// TwinCAT 3 PLC project PLC
// ProgramVersion: 3.1.4024.0
// libraries:
//   SPT Base Types, * (Beckhoff Automation LLC)
//   SPT Motion Control, * (Beckhoff Automation LLC)
//   Tc2_MC2, * (Beckhoff Automation GmbH)
//   Tc2_MC2_Drive, * (Beckhoff Automation GmbH)
//   Tc2_Standard, * (Beckhoff Automation GmbH)
//   Tc2_System, * (Beckhoff Automation GmbH)
//   Tc3_Module, * (Beckhoff Automation GmbH)
// project tree:
//   DUTs/ MoveState_t.TcDUT
//   GVLs/ IO.TcGVL (not stored), SafetyGlobalVariableList.TcGVL (not stored)
//   / PlcTask.TcTTO, SafetyTask.TcTTO
//   POUs/ MAIN.TcPOU (not stored), TestAxis1.TcPOU, SAFETY.TcPOU (not stored), TestAxis2.TcPOU
// real-time tasks:
//   TASK PlcTask: cycle T#10ms, priority 20, ADS port 350
//   TASK SafetyTask: cycle T#10ms, priority 21, ADS port 351
// motion (NC):
//   TASK NC-Task SAF: cycle T#2ms, priority 4, ADS port 501
//   TASK NC-Task SVB: cycle T#10ms, priority 8, ADS port 511
//   AXIS Axis 1 (id 1)
//     Dynamic: Acceleration=3272.24, Deceleration=3272.24, Jerk=9816.73
//     Velo: RefSearch=21.81495, RefSync=21.81495, SlowManual=109.07475, FastManual=654.4485, Fast=2181.495, Maximum=2181.49
//     PositionAreaControl: Enable=false, Range=1000
//     TargetPosControl: Enable=false, Range=1000
//     OtherSettings: AllowMotionCmdToSlave=true
//     encoder EncType=8
//       EncPara: ScaleFactorNumerator=60, ScaleFactorDenominator=1048576, MaxCount=#xffffffff
//     drive DrvType=9
//       DrvPara: MaxCount=#xffffffff, DriveControlDWord=#x00030100
//         Analog: VeloReferenz=2399.6445, VeloScale=1.02400649589962, TorqueSetpointScale=10, ScaleFactorActTorque=0.1
//         TimeComp: TaskDelayCycles=1
//     controller CtrType=1
//       CtrPara: PriorControlFactor=1
//         PosDiffControl: Enable=false, Range=15
//         Observer: BandWidth=20
//   AXIS Axis 2 (id 2)
//     Dynamic: Acceleration=3272.24, Deceleration=3272.24, Jerk=9816.73
//     Velo: RefSearch=21.81495, RefSync=21.81495, SlowManual=109.07475, FastManual=654.4485, Fast=2181.495, Maximum=2181.49
//     PositionAreaControl: Enable=false, Range=1000
//     TargetPosControl: Enable=false, Range=1000
//     OtherSettings: AllowMotionCmdToSlave=true
//     encoder EncType=8
//       EncPara: ScaleFactorNumerator=60, ScaleFactorDenominator=1048576, MaxCount=#xffffffff
//     drive DrvType=9
//       DrvPara: MaxCount=#xffffffff, DriveControlDWord=#x00030100
//         Analog: VeloReferenz=2399.6445, VeloScale=1.02400649589962, TorqueSetpointScale=10, ScaleFactorActTorque=0.1
//         TimeComp: TaskDelayCycles=1
//     controller CtrType=1
//       CtrPara: PriorControlFactor=1
//         PosDiffControl: Enable=false, Range=15
//         Observer: BandWidth=20
// I/O:
//   DEVICE CP6700-0001-0050, AmsNetId 5.81.155.22.4.1
//     Term 1 (EK1100) [EK1100 EtherCAT Coupler (2A E-Bus)]
//       Term 2 (EL1008) [EL1008 8Ch. Dig. Input 24V, 3ms]
//       Term 3 (EL1008) [EL1008 8Ch. Dig. Input 24V, 3ms]
//       Term 4 (EL2008) [EL2008 8Ch. Dig. Output 24V, 0.5A]
//       Term 5 (EL6910) [EL6910, TwinSAFE PLC]
//       Term 6 (EL1918) [EL1918, 8Ch. Safety Input 24V, TwinSAFE]
//         modules: Module 1 (FSOE), Module 2 (FSLOGIC)
//       Term 7 (EL2904) [EL2904, 4 Ch. Safety Output 24V, 0.5A, TwinSAFE]
//         modules: Module 1 (FSOES), Module 2 (DO)
//       Term 10 (EL9011) [EL9011 End Terminal]
//     Drive 8 (AX5206-0000-0213) [AX5206-0000-0213 EtherCAT Drive (SoE, 2 Ch.)]
//       Term 9 (AX5805) [AX5805 (Safety Drive Option)]
//         modules: Module 1 (Safety Process Data, 2 axis), Module 2 (Standard Process Data, 2 axis)
// variable links:
//   CP6700-0001-0050 <-> CP6700-0001-0050/Drive 8 (AX5206-0000-0213)/Term 9 (AX5805)
//     Term 1 (EK1100)/Term 5 (EL6910)/ConnectionInputs/TwinSafeGroup1.AX5805_4 TxPDO <-> Module 1 (Safety Process Data, 2 axis)/Outputs (Controlword)/FSOE
//   CP6700-0001-0050 <-> CP6700-0001-0050/Term 1 (EK1100)/Term 5 (EL6910)
//     Drive 8 (AX5206-0000-0213)/Term 9 (AX5805)/Module 1 (Safety Process Data, 2 axis)/Inputs (Statusword)/FSOE <-> ConnectionOutputs/TwinSafeGroup1.AX5805_4 RxPDO
//     Term 1 (EK1100)/Term 6 (EL1918)/Module 1 (FSOE)/FSoE Inputs/FSOE <-> ConnectionOutputs/TwinSafeGroup1.EL1918_2 RxPDO
//     Term 1 (EK1100)/Term 6 (EL1918)/Module 1 (FSOE)/FSoE Outputs/FSOE <-> ConnectionInputs/TwinSafeGroup1.EL1918_2 TxPDO
//   NC-Task SAF/Axes/Axis 1 <-> CP6700-0001-0050/Drive 8 (AX5206-0000-0213)
//     Drive/Inputs/In/nDataIn1 <-> AT 1/Following distance
//     Drive/Inputs/In/nDcOutputTime <-> InfoData/DcOutputShift
//     Drive/Inputs/In/nState1 <-> AT 1/Drive status word @bit 8
//     Drive/Inputs/In/nState2 <-> AT 1/Drive status word
//     Drive/Inputs/In/nState4 @bit 1 <-> WcState/InputToggle
//     Drive/Inputs/In/nState4 <-> WcState/WcState
//     Drive/Outputs/Out/nCtrl1 <-> MDT 1/Master control word @bit 8
//     Drive/Outputs/Out/nDataOut1 <-> MDT 1/Position command value
//     Enc/Inputs/In/nDataIn1 <-> AT 1/Position feedback 1 value
//     Enc/Inputs/In/nDcInputTime <-> InfoData/DcInputShift
//     Enc/Inputs/In/nState4 @bit 1 <-> WcState/InputToggle
//     Enc/Inputs/In/nState4 <-> WcState/WcState
//   NC-Task SAF/Axes/Axis 2 <-> CP6700-0001-0050/Drive 8 (AX5206-0000-0213)
//     Drive/Inputs/In/nDataIn1 <-> AT 2/Following distance
//     Drive/Inputs/In/nDcOutputTime <-> InfoData/DcOutputShift
//     Drive/Inputs/In/nState1 <-> AT 2/Drive status word @bit 8
//     Drive/Inputs/In/nState2 <-> AT 2/Drive status word
//     Drive/Inputs/In/nState4 @bit 1 <-> WcState/InputToggle
//     Drive/Inputs/In/nState4 <-> WcState/WcState
//     Drive/Outputs/Out/nCtrl1 <-> MDT 2/Master control word @bit 8
//     Drive/Outputs/Out/nDataOut1 <-> MDT 2/Position command value
//     Enc/Inputs/In/nDataIn1 <-> AT 2/Position feedback 1 value
//     Enc/Inputs/In/nDcInputTime <-> InfoData/DcInputShift
//     Enc/Inputs/In/nState4 @bit 1 <-> WcState/InputToggle
//     Enc/Inputs/In/nState4 <-> WcState/WcState
//   PLC/PLC Instance <-> CP6700-0001-0050/Term 1 (EK1100)/Term 2 (EL1008)
//     PlcTask Inputs/IO.DI4 <-> Channel 4/Input
//     SafetyTask Inputs/IO.DI1 <-> Channel 1/Input
//     SafetyTask Inputs/IO.DI2 <-> Channel 2/Input
//     SafetyTask Inputs/IO.DI3 <-> Channel 3/Input
//     SafetyTask Inputs/IO.DI5 <-> Channel 5/Input
//     SafetyTask Inputs/IO.DI6 <-> Channel 6/Input
//     SafetyTask Inputs/IO.DI7 <-> Channel 7/Input
//     SafetyTask Inputs/IO.DI8 <-> Channel 8/Input
//   PLC/PLC Instance <-> CP6700-0001-0050/Term 1 (EK1100)/Term 5 (EL6910)
//     PlcTask Inputs/SafetyGlobalVariableList.SAFETY_Permission <-> StandardInputs/TwinSafeGroup1.PLC_SAFETY_Permission_17
//     SafetyTask Inputs/SafetyGlobalVariableList.AX5805_Error_Ch1 <-> StandardInputs/TwinSafeGroup1.PLC_AX5805_Error_Ch1_13
//     SafetyTask Inputs/SafetyGlobalVariableList.AX5805_Error_Ch2 <-> StandardInputs/TwinSafeGroup1.PLC_AX5805_Error_Ch2_14
//     SafetyTask Inputs/SafetyGlobalVariableList.AX5805_STO_State_Ch1 <-> StandardInputs/TwinSafeGroup1.PLC_AX5805_STOState_Ch1_15
//     SafetyTask Inputs/SafetyGlobalVariableList.AX5805_STO_State_Ch2 <-> StandardInputs/TwinSafeGroup1.PLC_AX5805_STOState_Ch2_16
//     SafetyTask Inputs/SafetyGlobalVariableList.ERR_COM <-> StandardInputs/TwinSafeGroup1.ERR_COM_7
//     SafetyTask Inputs/SafetyGlobalVariableList.ERR_FB <-> StandardInputs/TwinSafeGroup1.ERR_FB_8
//     SafetyTask Inputs/SafetyGlobalVariableList.ERR_OTHER <-> StandardInputs/TwinSafeGroup1.ERR_OTHER_9
//     SafetyTask Inputs/SafetyGlobalVariableList.IN_RUN <-> StandardInputs/TwinSafeGroup1.IN_RUN_10
//     SafetyTask Outputs/SafetyGlobalVariableList.AX5805_ErrACK <-> StandardOutputs/TwinSafeGroup1.PLC_AX5805_ErrorAck_11
//     SafetyTask Outputs/SafetyGlobalVariableList.ERR_ACK <-> StandardOutputs/TwinSafeGroup1.ERR_ACK_5
//     SafetyTask Outputs/SafetyGlobalVariableList.RUN_STOP <-> StandardOutputs/TwinSafeGroup1.RUN_STOP_6
//     SafetyTask Outputs/SafetyGlobalVariableList.RestartFBs_TSG <-> StandardOutputs/TwinSafeGroup1.PLC_RestartFBs_12
//   PLC/PLC Instance <-> NC-Task SAF/Axes/Axis 2
//     PlcTask Inputs/MAIN.GoGoAxis2.AxisSPT._Axis.NcToPlc <-> Outputs/ToPlc
//     PlcTask Outputs/MAIN.GoGoAxis2.AxisSPT._Axis.PlcToNc <-> Inputs/FromPlc

CONFIGURATION PLC
    RESOURCE PLC ON TwinCAT3
        TASK PlcTask(INTERVAL := T#10ms, PRIORITY := 20);
        TASK SafetyTask(INTERVAL := T#10ms, PRIORITY := 21);
        PROGRAM MAIN WITH PlcTask : MAIN;
        PROGRAM SAFETY WITH SafetyTask : SAFETY;
    END_RESOURCE
END_CONFIGURATION

// ---- DUTs/MoveState_t.TcDUT
TYPE MoveState_t :
(
	MOVESTATE_INIT,
	MOVESTATE_ENABLE,
	MOVESTATE_FORWARD,
	MOVESTATE_BACKWARDS,
	MOVESTATE_BACKWARDSSLOW,
	MOVESTATE_NEWTARGETPOSITION,
	MOVESTATE_ERROR,
	MOVESTATE_RESET
);
END_TYPE

// ---- POUs/TestAxis1.TcPOU
FUNCTION_BLOCK TestAxis1
VAR
	
//	Axis1 : AXIS_REF;
//	StateAxis1: MoveState_t;
//	PowerAxis1: MC_Power;
//	Move_Y_MC_Axis1: MC_MoveAbsolute;
//	Move_X_MC_Axis1: MC_MoveAbsolute;
//	ResetAxis1: MC_Reset;
//	HomeAxis1: MC_Home;

//	SoEReadAxis1 : FB_SoERead;
//	SoEResetAxis1 : FB_SoEReset;
	
//	MoveAbsoluteOut1: ST_McOutputs;		(* debug function block output data *)
//	PowerAxis1Out: ST_McOutputs;		(* debug function block output data *)
//	MoveAbsoluteOut2: ST_McOutputs;		(* debug function block output data *)
//	ResetOut : ST_McOutputs;			(* debug function block output data *)

END_VAR

//	(* update the axis status at the beginning of each cycle *)
//		Axis1.ReadStatus();
//		SoEReadAxis1(Axis := Axis1);
//		SoEResetAxis1(Axis := Axis1);
//		PowerAxis1(Axis := Axis1);
//		ResetAxis1(Axis := Axis1);
//		Move_X_MC_Axis1(Axis := Axis1);
//		Move_Y_MC_Axis1(Axis := Axis1);
//		HomeAxis1(Axis := Axis1, bCalibrationCam := IO.DI4);

////IF SafetyGlobalVariableList.SAFETY_Permission = FALSE THEN

//// resetSafety();

////END_IF		
		
		
//IF SafetyGlobalVariableList.SAFETY_Permission = TRUE THEN

	
//	(* move axis using a state machine *)
//	CASE StateAxis1 OF

//		MOVESTATE_INIT :	(* initialisation *)
//			(* initialize all function blocks *)
//			Move_X_MC_Axis1.Execute	:= FALSE;
//			Move_Y_MC_Axis1.Execute	:= FALSE;
//			ResetAxis1.Execute		:= FALSE;
//			SoEResetAxis1.Execute 	:= FALSE;
//			StateAxis1				:= MOVESTATE_ENABLE;

//		MOVESTATE_ENABLE :
//			PowerAxis1.Enable := TRUE;
//			PowerAxis1.Enable_Positive := TRUE;
//			PowerAxis1.Enable_Negative := TRUE;
//			HomeAxis1.Execute := TRUE;

//			IF PowerAxis1.Status AND HomeAxis1.Done THEN
//				StateAxis1 := MOVESTATE_FORWARD;
//			ELSIF PowerAxis1.Error THEN
//				StateAxis1 := MOVESTATE_ERROR;
//			END_IF

//		MOVESTATE_FORWARD :		(* start to first position *)
//			Move_X_MC_Axis1.Position := 1500;		(* start to intermediate tartet position *)
//			Move_X_MC_Axis1.Velocity := 1500;		(* medium velocity level *)
//			Move_X_MC_Axis1.BufferMode := MC_Buffered;
//			Move_X_MC_Axis1.Execute := TRUE;
//			IF Move_X_MC_Axis1.Active  THEN
//				(* axis is executing job but is not yet finished *)
//				Move_X_MC_Axis1.Execute := FALSE;
//				(* leave this state and buffer a second command *)
//				StateAxis1 := MOVESTATE_NEWTARGETPOSITION;
//			ELSIF Move_X_MC_Axis1.CommandAborted OR Move_X_MC_Axis1.Error THEN
//				StateAxis1 := MOVESTATE_ERROR;
//			END_IF

//		MOVESTATE_NEWTARGETPOSITION :		(* change target position while moving *)
//			(* start a buffered motion command while axis is moving *)
//			Move_Y_MC_Axis1.Position := 5000;		(* start to final target *)
//			Move_Y_MC_Axis1.Velocity := 2000;		(* increase velocity *)
//			Move_Y_MC_Axis1.BufferMode := MC_BlendingPrevious; 	(* use velocity of previous command till intermediate target position position *)
//			Move_Y_MC_Axis1.Execute := TRUE;
//			IF Move_Y_MC_Axis1.Done THEN
//				Move_Y_MC_Axis1.Execute := FALSE;
//				StateAxis1 := MOVESTATE_BACKWARDS;
//			ELSIF Move_Y_MC_Axis1.CommandAborted OR Move_Y_MC_Axis1.Error THEN
//				StateAxis1 := MOVESTATE_ERROR;
//			END_IF

//		MOVESTATE_BACKWARDS :	(* move back to initial position *)
//			Move_X_MC_Axis1.Position := 100;		(* position close to initial position *)
//			Move_X_MC_Axis1.Velocity := 50;		(* high velocity *)
//			Move_X_MC_Axis1.BufferMode := MC_Buffered;
//			Move_X_MC_Axis1.Execute := TRUE;
//			IF Move_X_MC_Axis1.Active THEN
//				(* axis is executing job but is not yet finished *)
//				Move_X_MC_Axis1.Execute := FALSE;
//				(* leave this state and buffer a second command *)
//				StateAxis1 := MOVESTATE_BACKWARDSSLOW;
//			ELSIF Move_X_MC_Axis1.CommandAborted OR Move_X_MC_Axis1.Error THEN
//				StateAxis1 := MOVESTATE_ERROR;
//			END_IF

//		MOVESTATE_BACKWARDSSLOW :	(* move back to initial position *)
//			(* start a buffered motion command while axis is moving *)
//			Move_Y_MC_Axis1.Position := 0;	(* back to initial position *)
//			Move_Y_MC_Axis1.Velocity := 50; 	(* slow velocity *)
//			Move_Y_MC_Axis1.BufferMode := MC_BlendingNext; 	(* use velocity from first target position *)
//			Move_Y_MC_Axis1.Execute := TRUE;
//			IF Move_Y_MC_Axis1.Done THEN
//				Move_Y_MC_Axis1.Execute := FALSE;
//				StateAxis1 := MOVESTATE_FORWARD;
//			ELSIF Move_Y_MC_Axis1.CommandAborted OR Move_Y_MC_Axis1.Error THEN
//				StateAxis1 := MOVESTATE_ERROR;
//			END_IF

//		MOVESTATE_ERROR :
//			IF Axis1.Status.Error OR SoEReadAxis1.Error THEN
//				StateAxis1 := MOVESTATE_RESET;	(* axis error re quires reset *)
//			ELSE 
//				StateAxis1 := MOVESTATE_INIT;		(* function block errors don't need a reset *)
//			END_IF

//		MOVESTATE_RESET :
//			ResetAxis1.Execute := TRUE; 		
//			SoEResetAxis1.Execute := TRUE;
//			IF ResetAxis1.Done THEN
//				StateAxis1 := MOVESTATE_INIT;
//			ELSIF ResetAxis1.Error THEN
//				StateAxis1 := MOVESTATE_INIT; (* can't do anything here *)
//			END_IF

//	END_CASE

//END_IF

END_FUNCTION_BLOCK

// ---- POUs/TestAxis2.TcPOU
FUNCTION_BLOCK TestAxis2 EXTENDS FB_ComponentBase
VAR
	AxisSPT : FB_BasicAxis;
	State 	: INT;
END_VAR

METHOD PUBLIC CyclicLogic
VAR	

END_VAR
SUPER^.CyclicLogic();
END_METHOD

METHOD PROTECTED Initialize : BOOL;
SUPER^.Initialize();
END_METHOD

METHOD MoveAxis
      AxisSPT.CyclicLogic();

IF SafetyGlobalVariableList.SAFETY_Permission = TRUE THEN

	CASE State OF
		
	00:
		IF AxisSPT.Enable() THEN
			State := State + 10;
		END_IF
	10:
		IF AxisSPT.Enabled THEN
			AxisSPT.MoveVelocity( -5, TRUE);	
		
			IF IO.DI4 = TRUE THEN
				AxisSPT.Home();
				State := State + 10;
			END_IF
		END_IF

	
	20:
		AxisSPT.Velocity := 10;
		IF AxisSPT.MoveAbsolute(5000, FALSE) THEN
			State := State + 10;
		END_IF

	30:
		IF NOT AxisSPT.Busy THEN
			State := State + 10;
		END_IF

	40:
		AxisSPT.Trace('****Done****'); 

	50:
		//

	END_CASE

END_IF
END_METHOD

END_FUNCTION_BLOCK
